# EPICS substitutions: ek9000App/Db/EL1722_mbbiDirect.substitutions
file EL1722.template
{       pattern
        {
                TERMINAL,

        }
        {
        }
}
